// TIA Portal project "foratura_ghiera_V18_1" (V18)

(* hardware
DEVICE "S71500/ET200MP station_1"  S7-1500 station
   slot 0: "Telaio di montaggio_0"  Rack  6ES7 590-1***0-0AA0
   slot 0: "PM 190W 120/230VAC"  PM 190W 120/230VAC  6EP1333-4BA00
   slot 1: "PLC_1"  CPU 1516-3 PN/DP  6ES7 516-3AN01-0AB0  V2.5
      slot 3: "Display CPU_1"  6ES7591-1BA00-0AA0
   slot 2: "DI 32x24VDC HF_1"  DI 32x24VDC HF  6ES7 521-1BL00-0AB0  V1.0
   slot 3: "DQ 32x24VDC/0.5A HF_1"  DQ 32x24VDC/0.5A HF  6ES7 522-1BL01-0AB0  V1.0
   slot 4: "AI 8xU/I/RTD/TC ST_1"  AI 8xU/I/RTD/TC ST  6ES7 531-7KF00-0AB0  V1.0
   slot 5: "AQ 4xU/I ST_1"  AQ 4xU/I ST  6ES7 532-5HD00-0AB0  V1.0
*)

// ===== PLC "PLC_1"  CPU 1516-3 PN/DP =====

VAR_GLOBAL   // PLC tag table "Tabella delle variabili standard"
   "a0" AT %I0.7 : Bool;
   "stop" AT %I0.1 : Bool;
   "iPuls8" AT %I1.2 : Bool;
   "iPuls4" AT %I1.1 : Bool;
   "oUtensileAvanti" AT %Q0.0 : Bool;
   "iPuls2" AT %I0.0 : Bool;
   "oUtensileIndietro" AT %Q0.1 : Bool;
   "p2" AT %I0.2 : Bool;
   "p1" AT %I0.3 : Bool;
   "a1" AT %I0.6 : Bool;
   "b0" AT %I0.5 : Bool;
   "b1" AT %I0.4 : Bool;
   "oTransloAvanti" AT %Q0.2 : Bool;
   "oTransloIndietro" AT %Q0.3 : Bool;
   "luce" AT %Q0.4 : Bool;
   "sens_sportello" AT %Q1.0 : Bool;
   "Tag_1" AT %M0.0 : Bool;
   "portasportello" AT %I1.0 : Bool;
   "Tag_2" AT %M0.1 : Bool;
   "Tag_3" AT %M0.2 : Bool;
   "Tag_4" AT %M8.0 : Bool;
   "Tag_5" AT %M9.0 : Bool;
   "Tag_6" AT %M10.0 : Bool;
   "Tag_7" AT %M11.0 : Bool;
   "Tag_8" AT %M12.0 : Bool;
   "Tag_9" AT %M1.0 : Bool;
   "Tag_10" AT %M0.5 : Bool;
   "Tag_11" AT %M0.3 : Bool;
   "Tag_12" AT %M0.4 : Bool;
   "Tag_13" AT %M0.6 : Bool;
   "Tag_14" AT %M0.7 : Bool;
   "Tag_15" AT %M7.0 : Bool;
   "autoritenuta8" AT %M9.1 : Bool;
   "autoritenuta4" AT %M9.2 : Bool;
   "autoritenuta2" AT %M9.3 : Bool;
   "Clock_Byte" AT %MB100 : Byte;
   "Clock_10Hz" AT %M100.0 : Bool;
   "Clock_5Hz" AT %M100.1 : Bool;
   "Clock_2.5Hz" AT %M100.2 : Bool;
   "Clock_2Hz" AT %M100.3 : Bool;
   "Clock_1.25Hz" AT %M100.4 : Bool;
   "Clock_1Hz" AT %M100.5 : Bool;
   "Clock_0.625Hz" AT %M100.6 : Bool;
   "Clock_0.5Hz" AT %M100.7 : Bool;
   "System_Byte" AT %MB101 : Byte;
   "FirstScan" AT %M101.0 : Bool;
   "DiagStatusUpdate" AT %M101.1 : Bool;
   "AlwaysTRUE" AT %M101.2 : Bool;
   "AlwaysFALSE" AT %M101.3 : Bool;
   "ledVerde" AT %Q0.5 : Bool;
   "ledRosso" AT %Q1.5 : Bool;
END_VAR

// folder: System blocks/Program resources

DATA_BLOCK "conta_2"   // DB1
{ S7_Optimized_Access := 'TRUE' }
AUTHOR : Simatic
FAMILY : IEC
NAME : CNTR
VERSION : 1.0
// stored: InstanceOfName IEC_COUNTER
"IEC_COUNTER"
BEGIN
END_DATA_BLOCK

DATA_BLOCK "Conta_4"   // DB2
{ S7_Optimized_Access := 'TRUE' }
AUTHOR : Simatic
FAMILY : IEC
NAME : CNTR
VERSION : 1.0
// stored: InstanceOfName IEC_COUNTER
"IEC_COUNTER"
BEGIN
END_DATA_BLOCK

DATA_BLOCK "conta_4.1"   // DB3
{ S7_Optimized_Access := 'TRUE' }
AUTHOR : Simatic
FAMILY : IEC
NAME : CNTR
VERSION : 1.0
// stored: InstanceOfName IEC_COUNTER
"IEC_COUNTER"
BEGIN
END_DATA_BLOCK

DATA_BLOCK "conta_4.2"   // DB4
{ S7_Optimized_Access := 'TRUE' }
AUTHOR : Simatic
FAMILY : IEC
NAME : CNTR
VERSION : 1.0
// stored: InstanceOfName IEC_COUNTER
"IEC_COUNTER"
BEGIN
END_DATA_BLOCK

// folder: (top level)

FUNCTION "2fori" : Void   // FC1, LAD
{ S7_Optimized_Access := 'TRUE' }
VERSION : 0.1
BEGIN

REGION Network 1
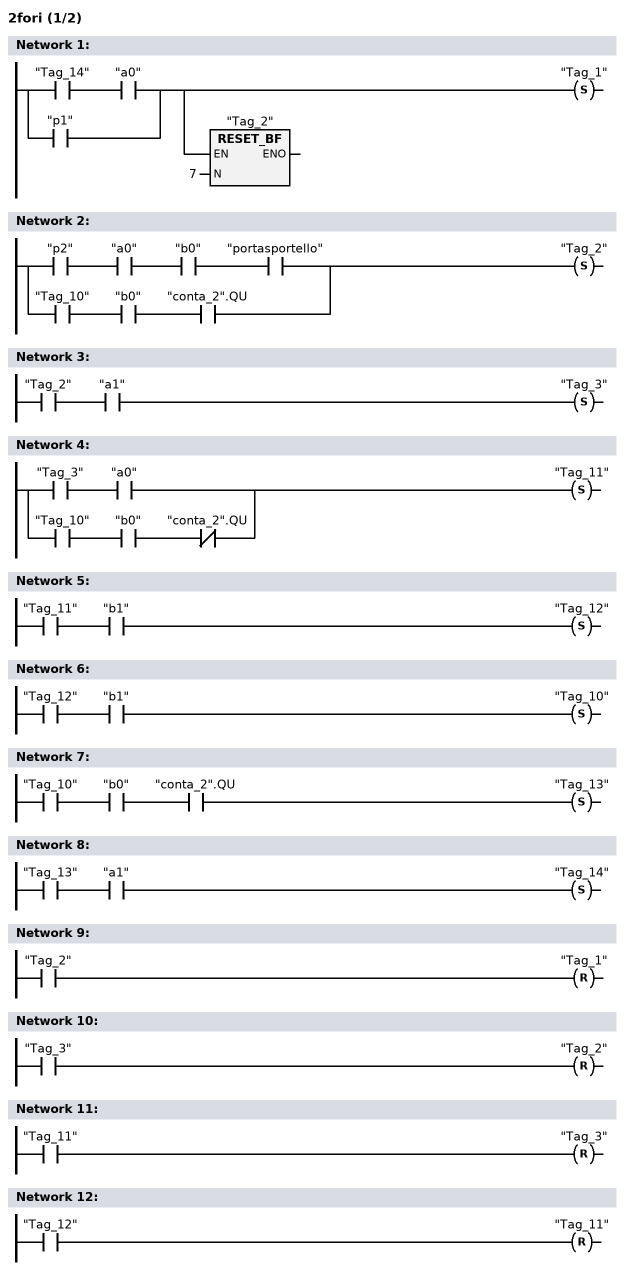
   // no SCL statement known for RBitfield: written as a call
   IF ("Tag_14" AND "a0") OR "p1" THEN
       "Tag_1" := TRUE;
       RESET_BF(operand := "Tag_2", n := 7);
   END_IF;
END_REGION

REGION Network 2
   RUNG wire#powerrail
      Contact( "p2" )
      Contact( "a0" )
      Contact( "b0" )
      Contact( "portasportello" )
      wire#w1
      S_Coil( "Tag_2" )
   END_RUNG
   RUNG wire#powerrail
      Contact( "Tag_10" )
      Contact( "b0" )
      Contact( "conta_2".QU )
   END_RUNG wire#w1
   // the same network as SCL:
   IF ("p2" AND "a0" AND "b0" AND "portasportello") OR ("Tag_10" AND "b0" AND "conta_2".QU) THEN
       "Tag_2" := TRUE;
   END_IF;
END_REGION

REGION Network 3
   RUNG wire#powerrail
      Contact( "Tag_2" )
      Contact( "a1" )
      S_Coil( "Tag_3" )
   END_RUNG
   // the same network as SCL:
   IF "Tag_2" AND "a1" THEN "Tag_3" := TRUE; END_IF;
END_REGION

REGION Network 4
   RUNG wire#powerrail
      Contact( "Tag_3" )
      Contact( "a0" )
      wire#w1
      S_Coil( "Tag_11" )
   END_RUNG
   RUNG wire#powerrail
      Contact( "Tag_10" )
      Contact( "b0" )
      I_Contact( "conta_2".QU )
   END_RUNG wire#w1
   // the same network as SCL:
   IF ("Tag_3" AND "a0") OR ("Tag_10" AND "b0" AND NOT "conta_2".QU) THEN "Tag_11" := TRUE; END_IF;
END_REGION

REGION Network 5
   RUNG wire#powerrail
      Contact( "Tag_11" )
      Contact( "b1" )
      S_Coil( "Tag_12" )
   END_RUNG
   // the same network as SCL:
   IF "Tag_11" AND "b1" THEN "Tag_12" := TRUE; END_IF;
END_REGION

REGION Network 6
   RUNG wire#powerrail
      Contact( "Tag_12" )
      Contact( "b1" )
      S_Coil( "Tag_10" )
   END_RUNG
   // the same network as SCL:
   IF "Tag_12" AND "b1" THEN "Tag_10" := TRUE; END_IF;
END_REGION

REGION Network 7
   RUNG wire#powerrail
      Contact( "Tag_10" )
      Contact( "b0" )
      Contact( "conta_2".QU )
      S_Coil( "Tag_13" )
   END_RUNG
   // the same network as SCL:
   IF "Tag_10" AND "b0" AND "conta_2".QU THEN "Tag_13" := TRUE; END_IF;
END_REGION

REGION Network 8
   RUNG wire#powerrail
      Contact( "Tag_13" )
      Contact( "a1" )
      S_Coil( "Tag_14" )
   END_RUNG
   // the same network as SCL:
   IF "Tag_13" AND "a1" THEN "Tag_14" := TRUE; END_IF;
END_REGION

REGION Network 9
   RUNG wire#powerrail
      Contact( "Tag_2" )
      R_Coil( "Tag_1" )
   END_RUNG
   // the same network as SCL:
   IF "Tag_2" THEN "Tag_1" := FALSE; END_IF;
END_REGION

REGION Network 10
   RUNG wire#powerrail
      Contact( "Tag_3" )
      R_Coil( "Tag_2" )
   END_RUNG
   // the same network as SCL:
   IF "Tag_3" THEN "Tag_2" := FALSE; END_IF;
END_REGION

REGION Network 11
   RUNG wire#powerrail
      Contact( "Tag_11" )
      R_Coil( "Tag_3" )
   END_RUNG
   // the same network as SCL:
   IF "Tag_11" THEN "Tag_3" := FALSE; END_IF;
END_REGION

REGION Network 12
   RUNG wire#powerrail
      Contact( "Tag_12" )
      R_Coil( "Tag_11" )
   END_RUNG
   // the same network as SCL:
   IF "Tag_12" THEN "Tag_11" := FALSE; END_IF;
END_REGION

REGION Network 13
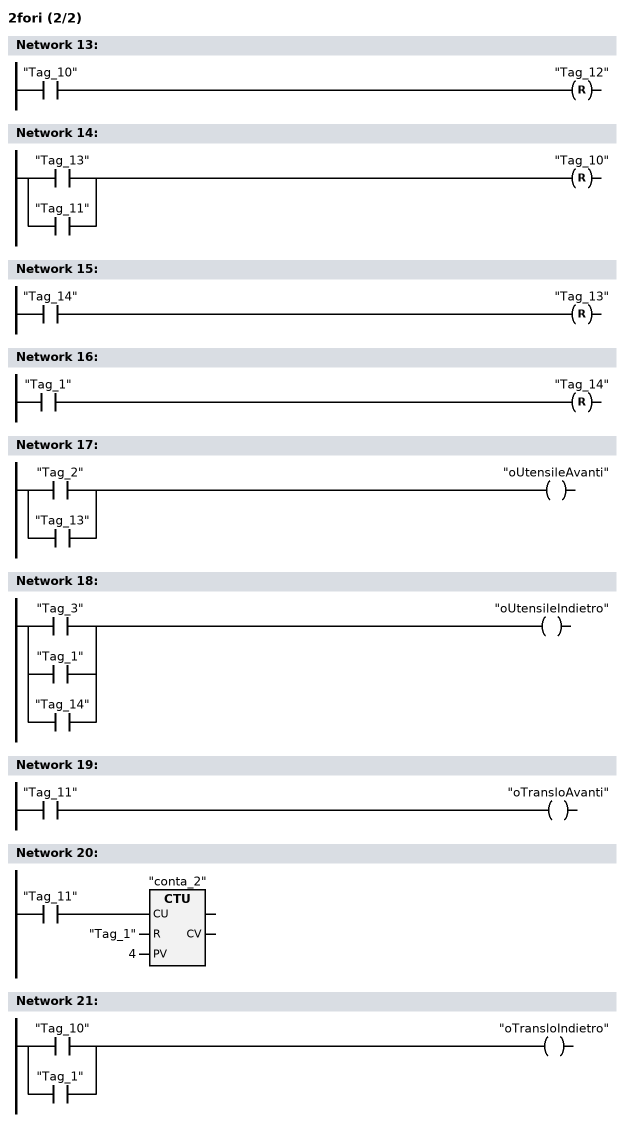
   RUNG wire#powerrail
      Contact( "Tag_10" )
      R_Coil( "Tag_12" )
   END_RUNG
   // the same network as SCL:
   IF "Tag_10" THEN "Tag_12" := FALSE; END_IF;
END_REGION

REGION Network 14
   RUNG wire#powerrail
      Contact( "Tag_13" )
      wire#w1
      R_Coil( "Tag_10" )
   END_RUNG
   RUNG wire#powerrail
      Contact( "Tag_11" )
   END_RUNG wire#w1
   // the same network as SCL:
   IF "Tag_13" OR "Tag_11" THEN "Tag_10" := FALSE; END_IF;
END_REGION

REGION Network 15
   RUNG wire#powerrail
      Contact( "Tag_14" )
      R_Coil( "Tag_13" )
   END_RUNG
   // the same network as SCL:
   IF "Tag_14" THEN "Tag_13" := FALSE; END_IF;
END_REGION

REGION Network 16
   RUNG wire#powerrail
      Contact( "Tag_1" )
      R_Coil( "Tag_14" )
   END_RUNG
   // the same network as SCL:
   IF "Tag_1" THEN "Tag_14" := FALSE; END_IF;
END_REGION

REGION Network 17
   RUNG wire#powerrail
      Contact( "Tag_2" )
      wire#w1
      Coil( "oUtensileAvanti" )
   END_RUNG
   RUNG wire#powerrail
      Contact( "Tag_13" )
   END_RUNG wire#w1
   // the same network as SCL:
   "oUtensileAvanti" := "Tag_2" OR "Tag_13";
END_REGION

REGION Network 18
   RUNG wire#powerrail
      Contact( "Tag_3" )
      wire#w1
      Coil( "oUtensileIndietro" )
   END_RUNG
   RUNG wire#powerrail
      Contact( "Tag_1" )
   END_RUNG wire#w1
   RUNG wire#powerrail
      Contact( "Tag_14" )
   END_RUNG wire#w1
   // the same network as SCL:
   "oUtensileIndietro" := "Tag_3" OR "Tag_1" OR "Tag_14";
END_REGION

REGION Network 19
   RUNG wire#powerrail
      Contact( "Tag_11" )
      Coil( "oTransloAvanti" )
   END_RUNG
   // the same network as SCL:
   "oTransloAvanti" := "Tag_11";
END_REGION

REGION Network 20
   "conta_2".CTU(CU := "Tag_11", R := "Tag_1", PV := 4);
END_REGION

REGION Network 21
   RUNG wire#powerrail
      Contact( "Tag_10" )
      wire#w1
      Coil( "oTransloIndietro" )
   END_RUNG
   RUNG wire#powerrail
      Contact( "Tag_1" )
   END_RUNG wire#w1
   // the same network as SCL:
   "oTransloIndietro" := "Tag_10" OR "Tag_1";
END_REGION
END_FUNCTION

FUNCTION "Blocco_1" : Void   // FC2, SCL
{ S7_Optimized_Access := 'TRUE' }
VERSION : 0.1
BEGIN
   IF "Tag_4" AND "a0" AND "conta_4.2".QU THEN
       "Tag_1" := TRUE;  
   END_IF;

   IF "p1" THEN
       "Tag_2" := TRUE;  
   END_IF;

   IF "p2" AND "a0" AND "b0" AND "portasportello" THEN
       "Tag_2" := TRUE;  
   END_IF;

   IF "Tag_10" AND "b0" AND "conta_2".QU THEN
       "Tag_2" := TRUE;  
   END_IF;

   IF "Tag_2" = 1 AND "a1" = 1 THEN
       "Tag_3" := 1;
   ELSE
       "Tag_3" := 0;
   END_IF;

   IF ("Tag_3" = 1 AND "a0" = 1) OR ("Tag_10" = 1 AND "b0" = 1 AND "conta_2".QU = 1) THEN
       "Tag_11" := 1;
   ELSE
       "Tag_11" := 0;
   END_IF;

   IF "Tag_11" THEN
       "luce" := TRUE;  
   ELSE
       "luce" := FALSE; 
   END_IF;


   IF ("Tag_12" AND "luce") THEN
       "Tag_10" := TRUE;  
   ELSE
       "Tag_10" := FALSE; 
   END_IF;


   IF ("Tag_10" AND "ledVerde" AND "conta_2".CU) THEN
       "Tag_13" := TRUE; 
   ELSE
       "Tag_13" := FALSE; 
   END_IF;

   // Segmento 8: SET di Tag_14
   IF "Tag_13" AND "a1" THEN
       "Tag_14" := TRUE;  // Set di Tag_14
   END_IF;

   // Segmento 9: RESET di Tag_1
   IF "Tag_2" THEN
       "Tag_1" := FALSE;  // Reset di Tag_1
   END_IF;

   // Segmento 10: RESET di Tag_2
   IF "Tag_3" THEN
       "Tag_2" := FALSE;  // Reset di Tag_2
   END_IF;

   // Segmento 11: RESET di Tag_3
   IF "Tag_11" THEN
       "Tag_3" := FALSE;  // Reset di Tag_3
   END_IF;

   // Segmento 12: RESET di Tag_11
   IF "Tag_12" THEN
       "Tag_11" := FALSE;  // Reset di Tag_11
   END_IF;

   // Segmento 13: RESET di Tag_12
   IF "Tag_10" THEN
       "Tag_12" := FALSE;  // Reset di Tag_12
   END_IF;

   IF ("Tag_13" OR "Tag_11") THEN
       "Tag_10" := FALSE;
   END_IF;


   IF "Tag_14" THEN
       "Tag_13" := FALSE;
   END_IF;

   IF "Tag_1" THEN
       "Tag_14" := FALSE;
   END_IF;

   IF "Tag_1" THEN
       "Tag_14" := FALSE; // Resetta M0.7
   END_IF;

   IF ("Tag_2" AND "Tag_13") THEN
       "oUtensileAvanti" := TRUE; // Attiva Q0.0
   ELSE
       "oUtensileAvanti" := FALSE; // Disattiva Q0.0 se la condizione non è soddisfatta
   END_IF;

   // Segmento 18: Controllo di Q0.1 (UtensileIndietro)
   IF ("Tag_3" OR "Tag_1" OR "Tag_14") THEN
       "oUtensileIndietro" := TRUE;
   ELSE
       "oUtensileIndietro" := FALSE;
   END_IF;

   // Segmento 19: Controllo di Q0.2 (TransloAvanti)
   IF "Tag_11" THEN
       "oTransloAvanti" := TRUE;
   ELSE
       "oTransloAvanti" := FALSE;
   END_IF;

   // Segmento 20: Contatore CTU

   //VAR
   //Conta_2:
   //CTU;           // Blocco contatore standard
   //Tag_1:
   //Bool := FALSE; // Variabile di reset
   //Tag_11:
   //Bool := FALSE; // Variabile di incremento
   //END_VAR

   // Logica del contatore
   // IF "Tag_1" THEN
       "conta_2".CV := 0;    // Reset contatore
   //ELSE
     //  "conta_2"(CU := "Tag_11",
       //          R := "Tag_1"); // Incremento contatore
   //END_IF;


       IF ("Tag_10" AND ("Tag_1" OR "Tag_10")) THEN
           "oTransloIndietro" := TRUE;
       ELSE
           "oTransloIndietro" := FALSE;
       END_IF;
END_FUNCTION

FUNCTION "8 fori" : Void   // FC3, LAD
{ S7_Optimized_Access := 'TRUE' }
VERSION : 0.1
BEGIN

REGION Network 1
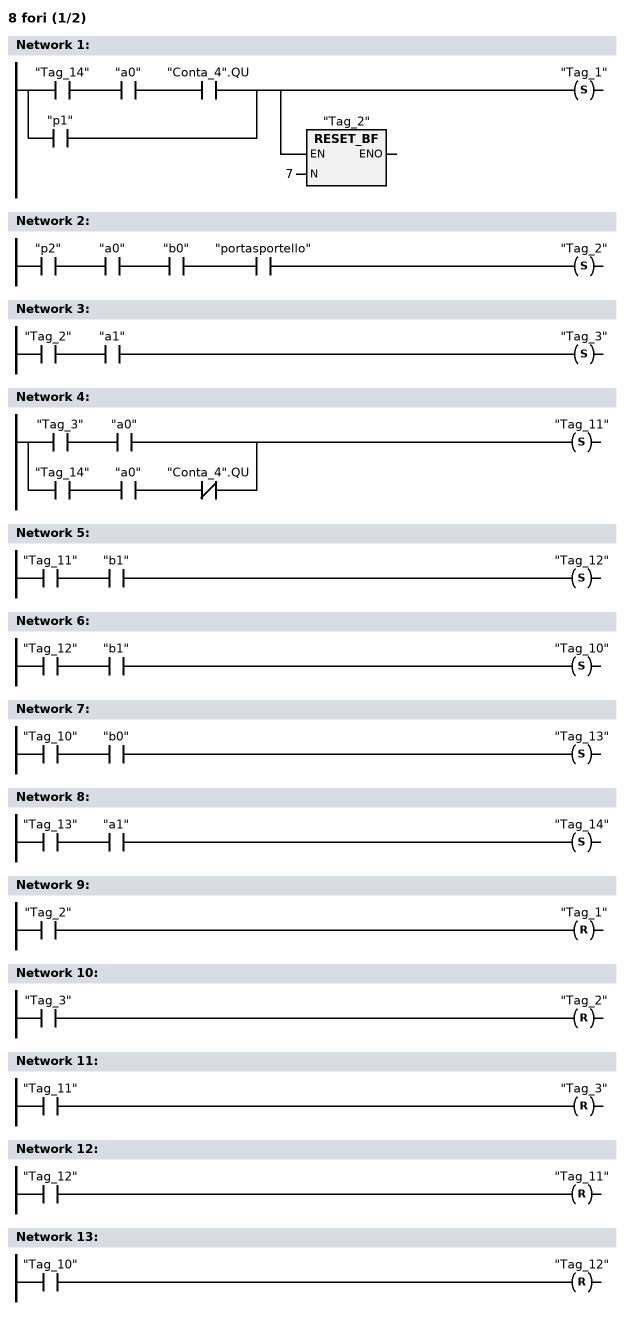
   // no SCL statement known for RBitfield: written as a call
   IF ("Tag_14" AND "a0" AND "Conta_4".QU) OR "p1" THEN
       "Tag_1" := TRUE;
       RESET_BF(operand := "Tag_2", n := 7);
   END_IF;
END_REGION

REGION Network 2
   RUNG wire#powerrail
      Contact( "p2" )
      Contact( "a0" )
      Contact( "b0" )
      Contact( "portasportello" )
      S_Coil( "Tag_2" )
   END_RUNG
   // the same network as SCL:
   IF "p2" AND "a0" AND "b0" AND "portasportello" THEN "Tag_2" := TRUE; END_IF;
END_REGION

REGION Network 3
   RUNG wire#powerrail
      Contact( "Tag_2" )
      Contact( "a1" )
      S_Coil( "Tag_3" )
   END_RUNG
   // the same network as SCL:
   IF "Tag_2" AND "a1" THEN "Tag_3" := TRUE; END_IF;
END_REGION

REGION Network 4
   RUNG wire#powerrail
      Contact( "Tag_3" )
      Contact( "a0" )
      wire#w1
      S_Coil( "Tag_11" )
   END_RUNG
   RUNG wire#powerrail
      Contact( "Tag_14" )
      Contact( "a0" )
      I_Contact( "Conta_4".QU )
   END_RUNG wire#w1
   // the same network as SCL:
   IF ("Tag_3" AND "a0") OR ("Tag_14" AND "a0" AND NOT "Conta_4".QU) THEN "Tag_11" := TRUE; END_IF;
END_REGION

REGION Network 5
   RUNG wire#powerrail
      Contact( "Tag_11" )
      Contact( "b1" )
      S_Coil( "Tag_12" )
   END_RUNG
   // the same network as SCL:
   IF "Tag_11" AND "b1" THEN "Tag_12" := TRUE; END_IF;
END_REGION

REGION Network 6
   RUNG wire#powerrail
      Contact( "Tag_12" )
      Contact( "b1" )
      S_Coil( "Tag_10" )
   END_RUNG
   // the same network as SCL:
   IF "Tag_12" AND "b1" THEN "Tag_10" := TRUE; END_IF;
END_REGION

REGION Network 7
   RUNG wire#powerrail
      Contact( "Tag_10" )
      Contact( "b0" )
      S_Coil( "Tag_13" )
   END_RUNG
   // the same network as SCL:
   IF "Tag_10" AND "b0" THEN "Tag_13" := TRUE; END_IF;
END_REGION

REGION Network 8
   RUNG wire#powerrail
      Contact( "Tag_13" )
      Contact( "a1" )
      S_Coil( "Tag_14" )
   END_RUNG
   // the same network as SCL:
   IF "Tag_13" AND "a1" THEN "Tag_14" := TRUE; END_IF;
END_REGION

REGION Network 9
   RUNG wire#powerrail
      Contact( "Tag_2" )
      R_Coil( "Tag_1" )
   END_RUNG
   // the same network as SCL:
   IF "Tag_2" THEN "Tag_1" := FALSE; END_IF;
END_REGION

REGION Network 10
   RUNG wire#powerrail
      Contact( "Tag_3" )
      R_Coil( "Tag_2" )
   END_RUNG
   // the same network as SCL:
   IF "Tag_3" THEN "Tag_2" := FALSE; END_IF;
END_REGION

REGION Network 11
   RUNG wire#powerrail
      Contact( "Tag_11" )
      R_Coil( "Tag_3" )
   END_RUNG
   // the same network as SCL:
   IF "Tag_11" THEN "Tag_3" := FALSE; END_IF;
END_REGION

REGION Network 12
   RUNG wire#powerrail
      Contact( "Tag_12" )
      R_Coil( "Tag_11" )
   END_RUNG
   // the same network as SCL:
   IF "Tag_12" THEN "Tag_11" := FALSE; END_IF;
END_REGION

REGION Network 13
   RUNG wire#powerrail
      Contact( "Tag_10" )
      R_Coil( "Tag_12" )
   END_RUNG
   // the same network as SCL:
   IF "Tag_10" THEN "Tag_12" := FALSE; END_IF;
END_REGION

REGION Network 14
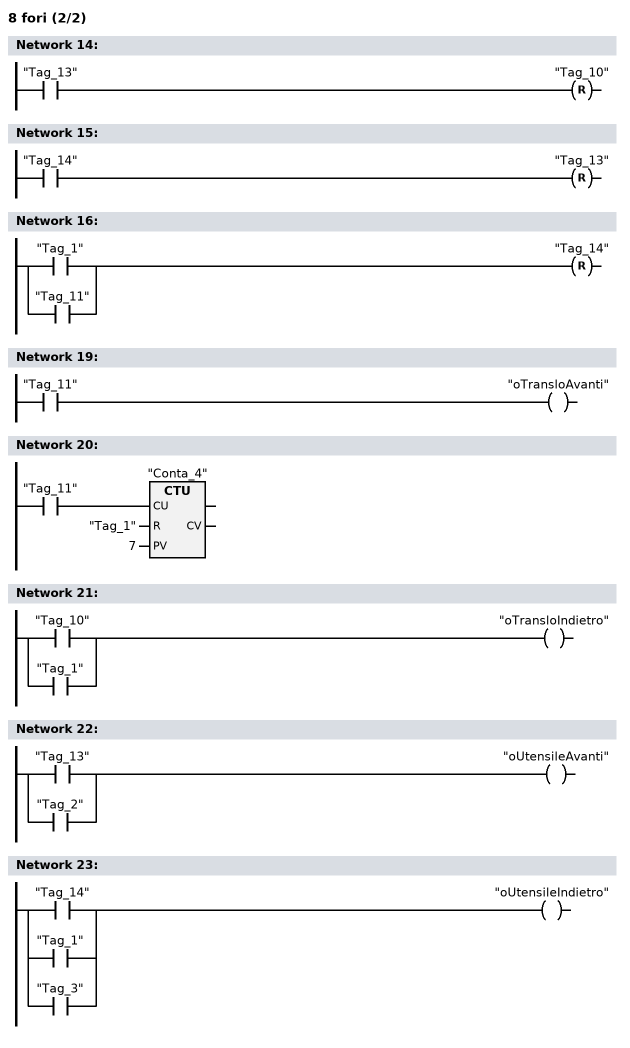
   RUNG wire#powerrail
      Contact( "Tag_13" )
      R_Coil( "Tag_10" )
   END_RUNG
   // the same network as SCL:
   IF "Tag_13" THEN "Tag_10" := FALSE; END_IF;
END_REGION

REGION Network 15
   RUNG wire#powerrail
      Contact( "Tag_14" )
      R_Coil( "Tag_13" )
   END_RUNG
   // the same network as SCL:
   IF "Tag_14" THEN "Tag_13" := FALSE; END_IF;
END_REGION

REGION Network 16
   RUNG wire#powerrail
      Contact( "Tag_1" )
      wire#w1
      R_Coil( "Tag_14" )
   END_RUNG
   RUNG wire#powerrail
      Contact( "Tag_11" )
   END_RUNG wire#w1
   // the same network as SCL:
   IF "Tag_1" OR "Tag_11" THEN "Tag_14" := FALSE; END_IF;
END_REGION

REGION Network 19
   RUNG wire#powerrail
      Contact( "Tag_11" )
      Coil( "oTransloAvanti" )
   END_RUNG
   // the same network as SCL:
   "oTransloAvanti" := "Tag_11";
END_REGION

REGION Network 20
   "Conta_4".CTU(CU := "Tag_11", R := "Tag_1", PV := 7);
END_REGION

REGION Network 21
   RUNG wire#powerrail
      Contact( "Tag_10" )
      wire#w1
      Coil( "oTransloIndietro" )
   END_RUNG
   RUNG wire#powerrail
      Contact( "Tag_1" )
   END_RUNG wire#w1
   // the same network as SCL:
   "oTransloIndietro" := "Tag_10" OR "Tag_1";
END_REGION

REGION Network 22
   RUNG wire#powerrail
      Contact( "Tag_13" )
      wire#w1
      Coil( "oUtensileAvanti" )
   END_RUNG
   RUNG wire#powerrail
      Contact( "Tag_2" )
   END_RUNG wire#w1
   // the same network as SCL:
   "oUtensileAvanti" := "Tag_13" OR "Tag_2";
END_REGION

REGION Network 23
   RUNG wire#powerrail
      Contact( "Tag_14" )
      wire#w1
      Coil( "oUtensileIndietro" )
   END_RUNG
   RUNG wire#powerrail
      Contact( "Tag_1" )
   END_RUNG wire#w1
   RUNG wire#powerrail
      Contact( "Tag_3" )
   END_RUNG wire#w1
   // the same network as SCL:
   "oUtensileIndietro" := "Tag_14" OR "Tag_1" OR "Tag_3";
END_REGION
END_FUNCTION

FUNCTION "4 fori" : Void   // FC4, LAD
{ S7_Optimized_Access := 'TRUE' }
VERSION : 0.1
BEGIN

REGION Network 1
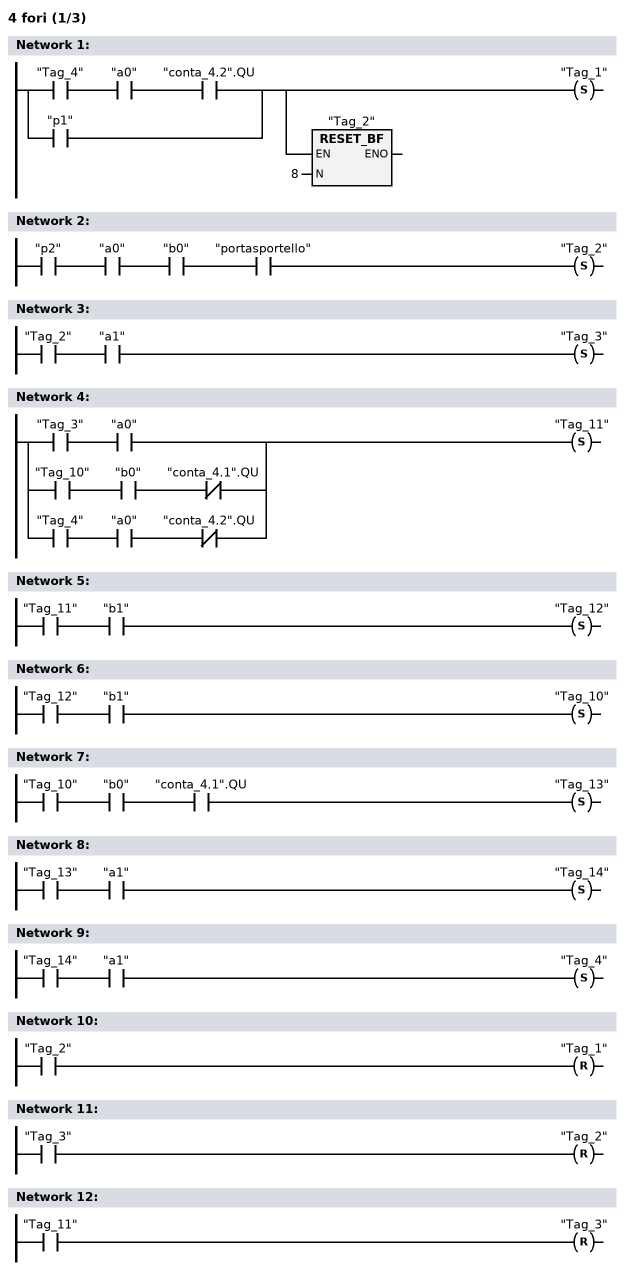
   // no SCL statement known for RBitfield: written as a call
   IF ("Tag_4" AND "a0" AND "conta_4.2".QU) OR "p1" THEN
       "Tag_1" := TRUE;
       RESET_BF(operand := "Tag_2", n := 8);
   END_IF;
END_REGION

REGION Network 2
   RUNG wire#powerrail
      Contact( "p2" )
      Contact( "a0" )
      Contact( "b0" )
      Contact( "portasportello" )
      S_Coil( "Tag_2" )
   END_RUNG
   // the same network as SCL:
   IF "p2" AND "a0" AND "b0" AND "portasportello" THEN "Tag_2" := TRUE; END_IF;
END_REGION

REGION Network 3
   RUNG wire#powerrail
      Contact( "Tag_2" )
      Contact( "a1" )
      S_Coil( "Tag_3" )
   END_RUNG
   // the same network as SCL:
   IF "Tag_2" AND "a1" THEN "Tag_3" := TRUE; END_IF;
END_REGION

REGION Network 4
   RUNG wire#powerrail
      Contact( "Tag_3" )
      Contact( "a0" )
      wire#w1
      S_Coil( "Tag_11" )
   END_RUNG
   RUNG wire#powerrail
      Contact( "Tag_10" )
      Contact( "b0" )
      I_Contact( "conta_4.1".QU )
   END_RUNG wire#w1
   RUNG wire#powerrail
      Contact( "Tag_4" )
      Contact( "a0" )
      I_Contact( "conta_4.2".QU )
   END_RUNG wire#w1
   // the same network as SCL:
   IF ("Tag_3" AND "a0") OR ("Tag_10" AND "b0" AND NOT "conta_4.1".QU) OR ("Tag_4" AND "a0" AND NOT "conta_4.2".QU) THEN
       "Tag_11" := TRUE;
   END_IF;
END_REGION

REGION Network 5
   RUNG wire#powerrail
      Contact( "Tag_11" )
      Contact( "b1" )
      S_Coil( "Tag_12" )
   END_RUNG
   // the same network as SCL:
   IF "Tag_11" AND "b1" THEN "Tag_12" := TRUE; END_IF;
END_REGION

REGION Network 6
   RUNG wire#powerrail
      Contact( "Tag_12" )
      Contact( "b1" )
      S_Coil( "Tag_10" )
   END_RUNG
   // the same network as SCL:
   IF "Tag_12" AND "b1" THEN "Tag_10" := TRUE; END_IF;
END_REGION

REGION Network 7
   RUNG wire#powerrail
      Contact( "Tag_10" )
      Contact( "b0" )
      Contact( "conta_4.1".QU )
      S_Coil( "Tag_13" )
   END_RUNG
   // the same network as SCL:
   IF "Tag_10" AND "b0" AND "conta_4.1".QU THEN "Tag_13" := TRUE; END_IF;
END_REGION

REGION Network 8
   RUNG wire#powerrail
      Contact( "Tag_13" )
      Contact( "a1" )
      S_Coil( "Tag_14" )
   END_RUNG
   // the same network as SCL:
   IF "Tag_13" AND "a1" THEN "Tag_14" := TRUE; END_IF;
END_REGION

REGION Network 9
   RUNG wire#powerrail
      Contact( "Tag_14" )
      Contact( "a1" )
      S_Coil( "Tag_4" )
   END_RUNG
   // the same network as SCL:
   IF "Tag_14" AND "a1" THEN "Tag_4" := TRUE; END_IF;
END_REGION

REGION Network 10
   RUNG wire#powerrail
      Contact( "Tag_2" )
      R_Coil( "Tag_1" )
   END_RUNG
   // the same network as SCL:
   IF "Tag_2" THEN "Tag_1" := FALSE; END_IF;
END_REGION

REGION Network 11
   RUNG wire#powerrail
      Contact( "Tag_3" )
      R_Coil( "Tag_2" )
   END_RUNG
   // the same network as SCL:
   IF "Tag_3" THEN "Tag_2" := FALSE; END_IF;
END_REGION

REGION Network 12
   RUNG wire#powerrail
      Contact( "Tag_11" )
      R_Coil( "Tag_3" )
   END_RUNG
   // the same network as SCL:
   IF "Tag_11" THEN "Tag_3" := FALSE; END_IF;
END_REGION

REGION Network 13
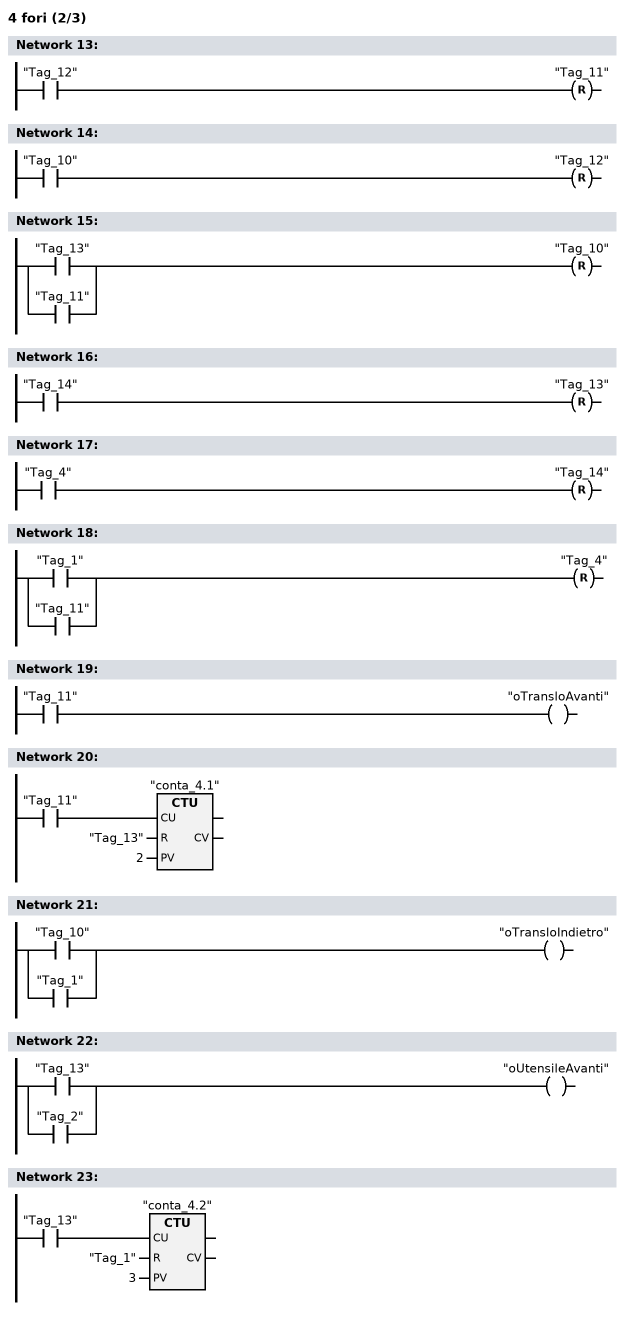
   RUNG wire#powerrail
      Contact( "Tag_12" )
      R_Coil( "Tag_11" )
   END_RUNG
   // the same network as SCL:
   IF "Tag_12" THEN "Tag_11" := FALSE; END_IF;
END_REGION

REGION Network 14
   RUNG wire#powerrail
      Contact( "Tag_10" )
      R_Coil( "Tag_12" )
   END_RUNG
   // the same network as SCL:
   IF "Tag_10" THEN "Tag_12" := FALSE; END_IF;
END_REGION

REGION Network 15
   RUNG wire#powerrail
      Contact( "Tag_13" )
      wire#w1
      R_Coil( "Tag_10" )
   END_RUNG
   RUNG wire#powerrail
      Contact( "Tag_11" )
   END_RUNG wire#w1
   // the same network as SCL:
   IF "Tag_13" OR "Tag_11" THEN "Tag_10" := FALSE; END_IF;
END_REGION

REGION Network 16
   RUNG wire#powerrail
      Contact( "Tag_14" )
      R_Coil( "Tag_13" )
   END_RUNG
   // the same network as SCL:
   IF "Tag_14" THEN "Tag_13" := FALSE; END_IF;
END_REGION

REGION Network 17
   RUNG wire#powerrail
      Contact( "Tag_4" )
      R_Coil( "Tag_14" )
   END_RUNG
   // the same network as SCL:
   IF "Tag_4" THEN "Tag_14" := FALSE; END_IF;
END_REGION

REGION Network 18
   RUNG wire#powerrail
      Contact( "Tag_1" )
      wire#w1
      R_Coil( "Tag_4" )
   END_RUNG
   RUNG wire#powerrail
      Contact( "Tag_11" )
   END_RUNG wire#w1
   // the same network as SCL:
   IF "Tag_1" OR "Tag_11" THEN "Tag_4" := FALSE; END_IF;
END_REGION

REGION Network 19
   RUNG wire#powerrail
      Contact( "Tag_11" )
      Coil( "oTransloAvanti" )
   END_RUNG
   // the same network as SCL:
   "oTransloAvanti" := "Tag_11";
END_REGION

REGION Network 20
   "conta_4.1".CTU(CU := "Tag_11", R := "Tag_13", PV := 2);
END_REGION

REGION Network 21
   RUNG wire#powerrail
      Contact( "Tag_10" )
      wire#w1
      Coil( "oTransloIndietro" )
   END_RUNG
   RUNG wire#powerrail
      Contact( "Tag_1" )
   END_RUNG wire#w1
   // the same network as SCL:
   "oTransloIndietro" := "Tag_10" OR "Tag_1";
END_REGION

REGION Network 22
   RUNG wire#powerrail
      Contact( "Tag_13" )
      wire#w1
      Coil( "oUtensileAvanti" )
   END_RUNG
   RUNG wire#powerrail
      Contact( "Tag_2" )
   END_RUNG wire#w1
   // the same network as SCL:
   "oUtensileAvanti" := "Tag_13" OR "Tag_2";
END_REGION

REGION Network 23
   "conta_4.2".CTU(CU := "Tag_13", R := "Tag_1", PV := 3);
END_REGION

REGION Network 24
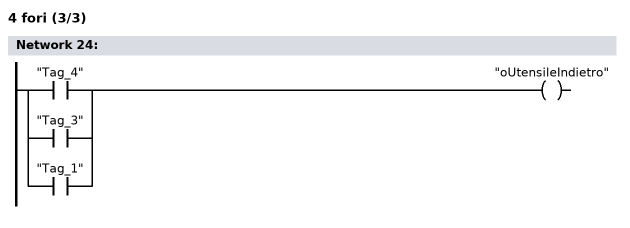
   RUNG wire#powerrail
      Contact( "Tag_4" )
      wire#w1
      Coil( "oUtensileIndietro" )
   END_RUNG
   RUNG wire#powerrail
      Contact( "Tag_3" )
   END_RUNG wire#w1
   RUNG wire#powerrail
      Contact( "Tag_1" )
   END_RUNG wire#w1
   // the same network as SCL:
   "oUtensileIndietro" := "Tag_4" OR "Tag_3" OR "Tag_1";
END_REGION
END_FUNCTION

ORGANIZATION_BLOCK "Main"   // OB1, LAD, ProgramCycle
TITLE = "Main Program Sweep (Cycle)"
{ S7_Optimized_Access := 'TRUE' }
VERSION : 0.1
   VAR_INPUT
      Initial_Call : Bool;   // Initial call of this OB
      Remanence : Bool;   // =True, if remanent data are available
   END_VAR
BEGIN

REGION Network 1
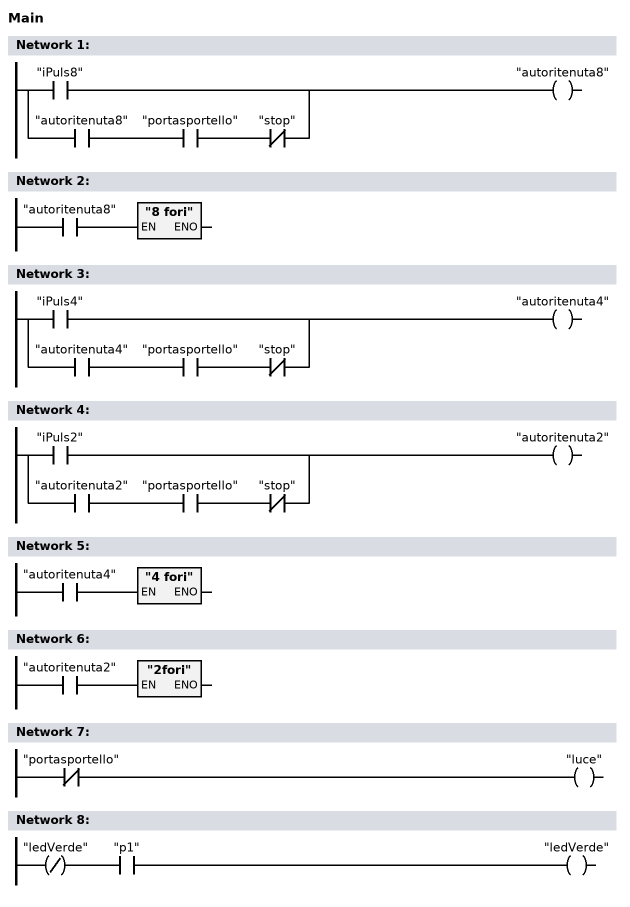
   RUNG wire#powerrail
      Contact( "iPuls8" )
      wire#w1
      Coil( "autoritenuta8" )
   END_RUNG
   RUNG wire#powerrail
      Contact( "autoritenuta8" )
      Contact( "portasportello" )
      I_Contact( "stop" )
   END_RUNG wire#w1
   // the same network as SCL:
   "autoritenuta8" := "iPuls8" OR ("autoritenuta8" AND "portasportello" AND NOT "stop");
END_REGION

REGION Network 2
   RUNG wire#powerrail
      Contact( "autoritenuta8" )
      "8 fori"()
   END_RUNG
   // the same network as SCL:
   IF "autoritenuta8" THEN "8 fori"(); END_IF;
END_REGION

REGION Network 3
   RUNG wire#powerrail
      Contact( "iPuls4" )
      wire#w1
      Coil( "autoritenuta4" )
   END_RUNG
   RUNG wire#powerrail
      Contact( "autoritenuta4" )
      Contact( "portasportello" )
      I_Contact( "stop" )
   END_RUNG wire#w1
   // the same network as SCL:
   "autoritenuta4" := "iPuls4" OR ("autoritenuta4" AND "portasportello" AND NOT "stop");
END_REGION

REGION Network 4
   RUNG wire#powerrail
      Contact( "iPuls2" )
      wire#w1
      Coil( "autoritenuta2" )
   END_RUNG
   RUNG wire#powerrail
      Contact( "autoritenuta2" )
      Contact( "portasportello" )
      I_Contact( "stop" )
   END_RUNG wire#w1
   // the same network as SCL:
   "autoritenuta2" := "iPuls2" OR ("autoritenuta2" AND "portasportello" AND NOT "stop");
END_REGION

REGION Network 5
   RUNG wire#powerrail
      Contact( "autoritenuta4" )
      "4 fori"()
   END_RUNG
   // the same network as SCL:
   IF "autoritenuta4" THEN "4 fori"(); END_IF;
END_REGION

REGION Network 6
   RUNG wire#powerrail
      Contact( "autoritenuta2" )
      "2fori"()
   END_RUNG
   // the same network as SCL:
   IF "autoritenuta2" THEN "2fori"(); END_IF;
END_REGION

REGION Network 7
   RUNG wire#powerrail
      I_Contact( "portasportello" )
      Coil( "luce" )
   END_RUNG
   // the same network as SCL:
   "luce" := NOT "portasportello";
END_REGION

REGION Network 8
   RUNG wire#powerrail
      I_Coil( "ledVerde" )
      Contact( "p1" )
      Coil( "ledVerde" )
   END_RUNG
   // the same network as SCL:
   "ledVerde" := NOT TRUE;
   "ledVerde" := "p1";
END_REGION
END_ORGANIZATION_BLOCK